(* IEC 61131-3 sources: TSA-FMICS22/ahorn/test/benchmark/arcade, 3 files *)

(* ---- 4.4.SafeMotionIO.st ---- *)
PROGRAM SafeMotionIO
USING PLCopenX;

  VAR_INPUT
	S1_S_EStopIn : SAFEBOOL;
    S2_S_AutoMode : SAFEBOOL;
    S2_S_SetupMode : SAFEBOOL;
    S4_S_EnableSwitchCh1 : SAFEBOOL;
    S4_S_EnableSwitchCh2 : SAFEBOOL;
    S5_S_GuardSwitch : SAFEBOOL;
    S7_S_GuardLock : SAFEBOOL;
    S0_Reset : BOOL;
    S8_UnlockGuard : BOOL;
    M1_S_AcknowledgeSS1 : SAFEBOOL;
    M1_S_AcknowledgeSafeMotion : SAFEBOOL;
  END_VAR
  VAR_OUTPUT
    S_SafeStop_M1 : SAFEBOOL;
    S_SafeMotion_M1 : SAFEBOOL;
    S_Enable_M1 : SAFEBOOL;
    S_UnlockGuard_K1 : SAFEBOOL;
  END_VAR
  VAR
    S_SetupMode : SAFEBOOL;
    S_AutoMode : SAFEBOOL;
    S_SafeStandstill : SAFEBOOL;
    S_SafeMotionActive : SAFEBOOL;
    SF_EmergencyStop_1 : SF_EmergencyStopX;
  	SF_SafetyRequest_1 : SF_SafetyRequestX;
  	SF_SafetyRequest_2 : SafetyRequest_dummy;
  	SF_ModeSelector_1 : SF_ModeSelectorX;
  	SF_GuardLocking_1 : SF_GuardLockingX;
  	SF_EnableSwitch_1 : SF_EnableSwitchX;
  END_VAR

  SF_EmergencyStop_1(TRUE, S1_S_EStopIn, FALSE, FALSE, S0_Reset);
  SF_SafetyRequest_1(TRUE, SF_EmergencyStop_1.S_EstopOut, M1_S_AcknowledgeSS1, T#100ms, S0_Reset);
  SF_SafetyRequest_2(TRUE, S_AutoMode, M1_S_AcknowledgeSafeMotion, T#100ms, S0_Reset);
  SF_ModeSelector_1(TRUE, S2_S_AutoMode, S2_S_SetupMode, FALSE, FALSE, FALSE, FALSE, FALSE, FALSE, TRUE, FALSE, TRUE, T#50ms, S0_Reset);
  SF_GuardLocking_1(TRUE, S5_S_GuardSwitch, S_SafeStandstill OR S_SafeMotionActive, S7_S_GuardLock, S8_UnlockGuard, FALSE, FALSE, S0_Reset);
  SF_EnableSwitch_1(TRUE, S_SafeMotionActive AND S_SetupMode, S4_S_EnableSwitchCh1, S4_S_EnableSwitchCh2, FALSE, S0_Reset);

  S_SafeStandstill := SF_SafetyRequest_1.S_SafetyActive;
  S_SafeStop_M1 := SF_SafetyRequest_1.S_SafetyRequest;
  S_SafeMotionActive := SF_SafetyRequest_2.S_SafetyActive;
  S_SafeMotion_M1 := SF_SafetyRequest_2.S_SafetyRequest;
  S_SetupMode := SF_ModeSelector_1.S_Mode1Sel;
  S_AutoMode := SF_ModeSelector_1.S_Mode0Sel AND SF_GuardLocking_1.S_GuardLocked;
  S_UnlockGuard_K1 := SF_GuardLocking_1.S_UnlockGuard;
  S_Enable_M1 := SF_EnableSwitch_1.S_EnableSwitchOut;

END_PROGRAM

FUNCTION_BLOCK SafetyRequest_dummy
VAR_INPUT
        Activate        : BOOL;
        S_OpMode        : SAFEBOOL;
        S_Acknowledge   : SAFEBOOL;
        MonitoringTime  : TIME := T#0s;
        Reset           : BOOL ;
 END_VAR

 VAR_OUTPUT
        Ready : BOOL ;
        S_SafetyActive : SAFEBOOL ;
        S_SafetyRequest : SAFEBOOL ;
        Error : BOOL ;
        DiagCode : WORD:=16#0000 ;
 END_VAR

VAR
        R_TRIGatReset: R_TRIG;
        T1: TONX;
END_VAR

R_TRIGatReset(CLK:=Reset);

IF NOT Activate THEN
    DiagCode := 16#0000;
ELSE

CASE DiagCode OF
16#0000:
    IF Activate THEN
        DiagCode := 16#8001;
    END_IF;
16#8000:
    IF NOT S_Acknowledge THEN
        DiagCode := 16#C002;
    ELSIF S_OpMode THEN
        DiagCode := 16#8012;
    END_IF;
16#8001:
    IF R_TRIGatReset.Q AND NOT S_Acknowledge THEN
        DiagCode := 16#8002;
    ELSIF R_TRIGatReset.Q AND S_Acknowledge THEN
        DiagCode := 16#8012;
    END_IF;
16#8002:
    IF NOT S_OpMode THEN
        DiagCode := 16#8003;
    ELSIF S_Acknowledge THEN
        DiagCode := 16#8012;
    END_IF;
16#8003:
    IF T1.Q THEN
        DiagCode := 16#C003;
    ELSIF S_OpMode THEN
        DiagCode := 16#8012;
    ELSIF S_Acknowledge THEN
        DiagCode := 16#8000;
    END_IF;
16#8005:
    IF S_OpMode THEN
        DiagCode := 16#8012;
    END_IF;
16#8012:
    IF NOT S_Acknowledge THEN
        DiagCode := 16#8002;
    ELSIF NOT S_OpMode THEN
        DiagCode := 16#8003;
    END_IF;
16#C002:
    IF Reset AND NOT R_TRIGatReset.Q THEN
        DiagCode := 16#C004;
    ELSIF R_TRIGatReset.Q THEN
        DiagCode := 16#8005;
    END_IF;
16#C003:
    IF Reset AND NOT R_TRIGatReset.Q THEN
        DiagCode := 16#C005;
    ELSIF R_TRIGatReset.Q THEN
        DiagCode := 16#8005;
    END_IF;
16#C004:
    IF NOT Reset THEN
        DiagCode := 16#C002;
    END_IF;
16#C005:
    IF NOT Reset THEN
        DiagCode := 16#C003;
    END_IF;
END_CASE;
END_IF;

IF DiagCode <> 16#8003 THEN
    T1(IN:=false, PT:=MonitoringTime);
ELSE
	T1(IN:=true, PT:=MonitoringTime);
END_IF;

CASE DiagCode OF
16#0000:
    Ready := FALSE;
    S_SafetyActive := FALSE;
    S_SafetyRequest := FALSE;
    Error := FALSE;
16#8000:
    Ready := TRUE;
    S_SafetyActive := TRUE;
    S_SafetyRequest := FALSE;
    Error := FALSE;
16#8001:
    Ready := TRUE;
    S_SafetyActive := FALSE;
    S_SafetyRequest := FALSE;
    Error := FALSE;
16#8002:
    Ready := TRUE;
    S_SafetyActive := FALSE;
    S_SafetyRequest := TRUE;
    Error := FALSE;
16#8003:
    Ready := TRUE;
    S_SafetyActive := FALSE;
    S_SafetyRequest := FALSE;
    Error := FALSE;
16#8005:
    Ready := TRUE;
    S_SafetyActive := FALSE;
    S_SafetyRequest := FALSE;
    Error := FALSE;
16#8012:
    Ready := TRUE;
    S_SafetyActive := FALSE;
    S_SafetyRequest := TRUE;
    Error := FALSE;
16#C002:
    Ready := TRUE;
    S_SafetyActive := FALSE;
    S_SafetyRequest := FALSE;
    Error := TRUE;
16#C003:
    Ready := TRUE;
    S_SafetyActive := FALSE;
    S_SafetyRequest := FALSE;
    Error := TRUE;
16#C004:
    Ready := TRUE;
    S_SafetyActive := FALSE;
    S_SafetyRequest := FALSE;
    Error := TRUE;
16#C005:
    Ready := TRUE;
    S_SafetyActive := FALSE;
    S_SafetyRequest := FALSE;
    Error := TRUE;
END_CASE;

END_FUNCTION_BLOCK;

(* ---- 4.1.DiagnosticsConcept.st ---- *)
PROGRAM DiagnosticsConcept
USING PLCopenX;

  VAR_INPUT
	S1_S_EStopIn_1 : SAFEBOOL;
	S1_S_EStopIn_2 : SAFEBOOL;
	S2_S_ESPE_In : SAFEBOOL;
	S0_Reset : BOOL;
	S3_Drive_Reset : BOOL;
	AxisD_1 : INT;
	InputDevice1_active : BOOL;
	InputDevice2_active : BOOL;
	Internal_Acknowledge: BOOL;
  END_VAR
  VAR_OUTPUT
    Error_Equiv1 : BOOL;
	Diag_Equiv1 : WORD;
	Error_EStop1 : BOOL;
	Diag_EStop1 : WORD;
	Error_ESPE1 : BOOL;
	Diag_ESPE1 : WORD;
	Error_SafeStop1 : BOOL;
	Diag_SafeStop1 : WORD;
    S_Stopped : BOOL;
  END_VAR
  VAR
  	S_EStopOut : SAFEBOOL;
	SF_Equivalent_1 : SF_EquivalentX;
	SF_EmergencyStop_1 : SF_EmergencyStopX;
	SF_ESPE_1 : SF_ESPEX;
	SF_SafeStop1_1 : SF_SafeStop1X;
  END_VAR

  SF_Equivalent_1(InputDevice1_active, S1_S_EStopIn_1, S1_S_EStopIn_2, T#10ms);
  SF_EmergencyStop_1(SF_Equivalent_1.Ready, SF_Equivalent_1.S_EquivalentOut, FALSE, FALSE, S0_Reset);
  SF_ESPE_1(InputDevice2_active, S2_S_ESPE_In, FALSE, FALSE, S0_Reset);
  SF_SafeStop1_1(
    Activate:=SF_EmergencyStop_1.Ready AND SF_ESPE_1.Ready,
    S_StopIn:=S_EStopOut AND SF_ESPE_1.S_ESPE_Out,
    AxisID:=AxisD_1,
    MonitoringTime:=T#100ms,
    Reset:=S3_Drive_Reset,
    Acknowledge := Internal_Acknowledge);
  S_EStopOut := SF_EmergencyStop_1.S_EStopOut;
  Error_Equiv1 := SF_Equivalent_1.Error;
  Diag_Equiv1 := SF_Equivalent_1.DiagCode;
  Error_EStop1 := SF_EmergencyStop_1.Error;
  Diag_EStop1 := SF_EmergencyStop_1.DiagCode;
  Error_ESPE1 := SF_ESPE_1.Error;
  Diag_ESPE1 := SF_ESPE_1.DiagCode;
  Error_SafeStop1 := SF_SafeStop1_1.Error;
  Diag_SafeStop1 := SF_SafeStop1_1.DiagCode;
  S_Stopped := SF_SafeStop1_1.S_Stopped;
END_PROGRAM

(* ---- RTAndroid_flagDelayAsInput.st ---- *)
PROGRAM cyclic
(* Moegliche Zustaende fuer den Automaten *)
VAR CONSTANT
	stateAfterBoot : BYTE := 0;
	stateInit : BYTE := 1;
	stateWaitForItem : BYTE := 2;
	stateWaitForCompressor1 : BYTE := 3;
	stateExtractItem1 : BYTE := 4;
	stateWaitForCompressor2 : BYTE := 5;
	stateExtractItem2 : BYTE := 6;
	stateRotateTable1 : BYTE := 7;
	stateWaitForCompressor3 : BYTE := 8;
	statePunchItem : BYTE := 9;
	stateRotateTable2 : BYTE := 10;
	stateWaitForCompressor4 : BYTE := 11;
	stateMoveToConveyer1 : BYTE := 12;
	stateWaitForCompressor5 : BYTE := 13;
	stateMoveToConveyer2 : BYTE := 14;
	stateRunConveyer : BYTE := 15;
	stateMoveToRobot : BYTE := 16;
	stateTurnToItem : BYTE := 17;
	stateTakeItem : BYTE := 18;
	stateTurnToMagazin : BYTE := 19;
	stateError : BYTE := 20;
END_VAR
(* Vordefinierte Konstanten fuer den gesamten Ablauf *)
VAR CONSTANT
	pickPosTurn : BYTE := 111;
	pickPosVert : BYTE := 80;
	pickPosArm : BYTE := 28;
	pickPosClaw : BYTE := 19;
	dropPosTurn : BYTE := 71;
	dropPosArm : BYTE := 37;
	moveThreshold : BYTE := 36;
	compressorDelay : DINT := 50;
	extractionDelay : DINT := 50;
	conveyerDelay : DINT := 50;
	waitForItemThreshold : DINT := 100;
	waitForPuncherThreshold : DINT := 10;
END_VAR
(* Virtuelle Speicherstellen der Sensoren / Motoren *)
VAR_INPUT
	(* 3D-Roboter *)
	turnDestPos : BYTE;
	turnCurrPos : BYTE;
	vertDestPos  : BYTE;
	vertCurrPos : BYTE;
	armDestPos  : BYTE;
	armCurrPos   : BYTE;
	clawDestPos  : BYTE;
	clawCurrPos  : BYTE;
	(* Bearbeitungszentrum *)
	compressor : BYTE;
	tableMotPow  : BYTE;
	tableMotDir  : BYTE;
	magazinLed  : BYTE;
	magazinPhoto : BYTE;
	magazinPusherOn  : BYTE;
	magazinPusherOff : BYTE;
	conveyerMotPow  : BYTE;
	conveyerMotDir  : BYTE;
	conveyerLed  : BYTE;
	conveyerPhoto  : BYTE;
	conveyerButton : BYTE;
	conveyerPusherOn  : BYTE;
	conveyerPusherOff  : BYTE;
	puncherButton  : BYTE;
	puncher  : BYTE;

	flagDelay : DINT;
END_VAR

(* Verwendete Ein- und Ausgaenge *)
VAR_OUTPUT
	outState : BYTE;
	outError : BOOL := false;
	DiagCode : BYTE := 16#0000;
END_VAR

	(* Motoren einmalig zur Nullposition fahren *)
	IF DiagCode = stateAfterBoot THEN

		compressor := 0;

		tableMotPow := 0;
		tableMotDir := 0;

		magazinLed := 0;
		magazinPusherOn := 0;
		magazinPusherOff := 0;

		conveyerMotPow := 0;
		conveyerMotDir := 0;
		conveyerLed := 0;
		conveyerPusherOn := 0;
		conveyerPusherOff := 0;

		turnDestPos := 0;
		vertDestPos := 0;
		armDestPos := 0;
		clawDestPos := 0;

		IF turnCurrPos = 0 AND armCurrPos = 0 AND clawCurrPos = 0 THEN
			DiagCode := stateInit;
		END_IF

	(* Anlage vor dem Start initialisieren *)
	ELSIF DiagCode = stateInit THEN

		conveyerLed := 1;
		magazinLed := 1;

		turnDestPos := dropPosTurn;
		armDestPos := dropPosArm;

		IF turnCurrPos = dropPosTurn AND armCurrPos = dropPosArm AND vertCurrPos = 0 THEN
			IF clawCurrPos = 0 THEN
				DiagCode := stateWaitForItem;
			ELSE
				clawDestPos := 0;
			END_IF
		END_IF

	(* Warten, bis sich ein Werkstueck im Magazin befindet *)
	ELSIF DiagCode = stateWaitForItem THEN

		IF flagDelay = waitForItemThreshold THEN
			DiagCode := stateInit;
		ELSIF magazinPhoto = 1 THEN
			magazinLed := 0;
			DiagCode := stateWaitForCompressor1;
		END_IF

	(* Kompressor zum Ausfahren des Magazinschiebers vorbereiten *)
	ELSIF DiagCode = stateWaitForCompressor1 THEN

		compressor := 1;

		IF flagDelay >= compressorDelay THEN
			compressor := 0;
			DiagCode := stateExtractItem1;
		END_IF

	(* Werkstueck aus dem Magazin entnehmen - Teil 1 *)
	ELSIF DiagCode = stateExtractItem1 THEN

		magazinPusherOn := 1;

		IF flagDelay >= extractionDelay THEN
			magazinPusherOn := 0;
			DiagCode := stateWaitForCompressor2;
		END_IF

	(* Kompressor zum Einfahren des Magazinschiebers vorbereiten *)
	ELSIF DiagCode = stateWaitForCompressor2 THEN

		compressor := 1;

		IF flagDelay >= compressorDelay THEN
			compressor := 0;
			DiagCode := stateExtractItem2;
		END_IF

	(* Werkstueck aus dem Magazin entnehmen - Teil 2 *)
	ELSIF DiagCode = stateExtractItem2 THEN

		magazinPusherOff := 1;

		IF flagDelay >= extractionDelay THEN
			magazinPusherOff := 0;
			DiagCode := stateRotateTable1;
		END_IF

	(* Drehtisch aktivieren und Stanze-Schalter ueberwachen *)
	ELSIF DiagCode = stateRotateTable1 THEN

		tableMotPow := 200;
		(* something went wrong: we skip punching *)
		IF flagDelay > waitForPuncherThreshold THEN
			tableMotPow := 0;
			DiagCode := stateRotateTable2;
		ELSIF puncherButton = 0 THEN
			tableMotPow := 0;
			DiagCode := stateWaitForCompressor3;
		END_IF

	(* Kompressor zum Stanzen vorbereiten *)
	ELSIF DiagCode = stateWaitForCompressor3 THEN

		compressor := 1;

		IF flagDelay >= compressorDelay THEN
			compressor := 0;
			DiagCode := statePunchItem;
		END_IF

	(* Werkstueck stanzen *)
	ELSIF DiagCode = statePunchItem THEN

		puncher := 1;

		IF flagDelay >= extractionDelay THEN
			puncher := 0;
			DiagCode := stateRotateTable2;
		END_IF

	(* Drehtisch aktivieren und Transportband-Schalter ueberwachen *)
	ELSIF DiagCode = stateRotateTable2 THEN

		tableMotPow := 200;

		IF conveyerButton = 0 THEN
			tableMotPow := 0;
			DiagCode := stateWaitForCompressor4;
		END_IF
	(* Kompressor zum Einfahren des Transportschiebers vorbereiten *)
	ELSIF DiagCode = stateWaitForCompressor4 THEN

		compressor := 1;

		IF flagDelay >= compressorDelay THEN
			compressor := 0;
			DiagCode := stateMoveToConveyer1;
		END_IF

	(* Werkstueck auf das Fliessband befoerdern - Teil 1 *)
	ELSIF DiagCode = stateMoveToConveyer1 THEN

		conveyerPusherOn := 1;

		IF flagDelay >= extractionDelay THEN
			conveyerPusherOn := 0;
			DiagCode := stateWaitForCompressor5;
		END_IF

	(* Kompressor zum Ausfahren des Transportschiebers vorbereiten *)
	ELSIF DiagCode = stateWaitForCompressor5 THEN

		compressor := 1;

		IF flagDelay >= compressorDelay THEN
			compressor := 0;
			DiagCode := stateMoveToConveyer2;
		END_IF

	(* Werkstueck auf das Fliessband befoerdern - Teil 2 *)
	ELSIF DiagCode = stateMoveToConveyer2 THEN

		conveyerPusherOff := 1;

		IF flagDelay >= extractionDelay THEN
			conveyerPusherOff := 0;
			DiagCode := stateRunConveyer;
		END_IF

	(* Fliessband aktivieren und auf das Werkstueck warten *)
	ELSIF DiagCode = stateRunConveyer THEN

		conveyerMotPow := 200;
		(*Something went wrong, we again try to put the item on the tape *)
		IF flagDelay = waitForItemThreshold THEN
			DiagCode := stateMoveToConveyer1;
		ELSIF conveyerPhoto = 1 THEN
			conveyerLed := 0;
			DiagCode := stateMoveToRobot;
		END_IF

	(* Drehen, Greifarm und Greifer ausstrecken *)
	ELSIF DiagCode = stateMoveToRobot THEN

		IF flagDelay > conveyerDelay THEN
			conveyerMotPow := 0;
			DiagCode := stateTurnToItem;
		END_IF

	(* Drehen, Greifarm und Greifer ausstrecken *)
	ELSIF DiagCode = stateTurnToItem THEN

		turnDestPos := pickPosTurn;
		vertDestPos := pickPosVert;
		armDestPos := pickPosArm;

		IF turnCurrPos = pickPosTurn AND vertCurrPos = pickPosVert AND armCurrPos = pickPosArm THEN
			DiagCode := stateTakeItem;
		END_IF

	(* Werkstueck vom Fliessband greifen *)
	ELSIF DiagCode = stateTakeItem THEN

		clawDestPos := pickPosClaw;

		IF clawCurrPos = pickPosClaw THEN
			DiagCode := stateTurnToMagazin;
		END_IF

	(* Das Werkstueck zum Magazin drehen *)
	ELSIF DiagCode = stateTurnToMagazin THEN

		vertDestPos := 0;

		IF vertCurrPos < moveThreshold THEN
			DiagCode := stateInit;
		END_IF

	(* Fehlerzustand - alles ausschalten *)
	ELSE

		outError := true;

		compressor := 0;
		puncher := 0;

		tableMotPow := 0;
		tableMotDir := 2;

		conveyerMotPow := 0;
		conveyerMotDir := 2;

	(* Ende des Zustandsautomaten *)
	END_IF

	(* Ausgabe vorbereiten *)
	outState := DiagCode;

END_PROGRAM
